TYPE DUT_HMI_Production_Counters :
STRUCT
	TotalPieceGood : UDINT;
	TotalPieceScrap : UDINT;
END_STRUCT
END_TYPE

(* stored: Version 1.1.0.1, ProductVersion 3.1.4024.15
   DUT DUT_HMI_Production_Counters: Id {2f9958b9-0c5e-4d8f-b3ca-39534ec6d113} *)
